FUNCTION LWORD_TO_QUARTERS
  (* Standard: 61499-1; Description: Copyright (c) 2024 HR Agrartechnik GmbH This program and the accompanying materials are made available under the terms of the Eclipse Public License 2.0 which is available at https://www.eclipse.org/legal/epl-2.0/ SPDX-License-Identifier: EPL-2.0 *)
  (* Version 1.0, 2024-02-22, franz *)
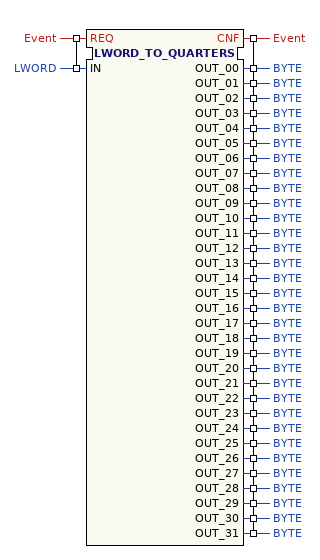
  EVENT_INPUT
    REQ WITH IN; (* Normal Execution Request *)
  END_EVENT
  EVENT_OUTPUT
    CNF WITH OUT_00, OUT_01, OUT_02, OUT_03, OUT_04, OUT_05, OUT_06, OUT_07, OUT_08, OUT_09, OUT_10, OUT_11, OUT_12, OUT_13, OUT_14, OUT_15, OUT_16, OUT_17, OUT_18, OUT_19, OUT_20, OUT_21, OUT_22, OUT_23, OUT_24, OUT_25, OUT_26, OUT_27, OUT_28, OUT_29, OUT_30, OUT_31; (* Execution Confirmation *)
  END_EVENT
  VAR_INPUT
    IN : LWORD; (* LWORD Input *)
  END_VAR
  VAR_OUTPUT
    OUT_00 : BYTE; (* QUARTER BYTE 00 *)
    OUT_01 : BYTE; (* QUARTER BYTE 01 *)
    OUT_02 : BYTE; (* QUARTER BYTE 02 *)
    OUT_03 : BYTE; (* QUARTER BYTE 03 *)
    OUT_04 : BYTE; (* QUARTER BYTE 04 *)
    OUT_05 : BYTE; (* QUARTER BYTE 05 *)
    OUT_06 : BYTE; (* QUARTER BYTE 06 *)
    OUT_07 : BYTE; (* QUARTER BYTE 07 *)
    OUT_08 : BYTE; (* QUARTER BYTE 08 *)
    OUT_09 : BYTE; (* QUARTER BYTE 09 *)
    OUT_10 : BYTE; (* QUARTER BYTE 10 *)
    OUT_11 : BYTE; (* QUARTER BYTE 11 *)
    OUT_12 : BYTE; (* QUARTER BYTE 12 *)
    OUT_13 : BYTE; (* QUARTER BYTE 13 *)
    OUT_14 : BYTE; (* QUARTER BYTE 14 *)
    OUT_15 : BYTE; (* QUARTER BYTE 15 *)
    OUT_16 : BYTE; (* QUARTER BYTE 16 *)
    OUT_17 : BYTE; (* QUARTER BYTE 17 *)
    OUT_18 : BYTE; (* QUARTER BYTE 18 *)
    OUT_19 : BYTE; (* QUARTER BYTE 19 *)
    OUT_20 : BYTE; (* QUARTER BYTE 20 *)
    OUT_21 : BYTE; (* QUARTER BYTE 21 *)
    OUT_22 : BYTE; (* QUARTER BYTE 22 *)
    OUT_23 : BYTE; (* QUARTER BYTE 23 *)
    OUT_24 : BYTE; (* QUARTER BYTE 24 *)
    OUT_25 : BYTE; (* QUARTER BYTE 25 *)
    OUT_26 : BYTE; (* QUARTER BYTE 26 *)
    OUT_27 : BYTE; (* QUARTER BYTE 27 *)
    OUT_28 : BYTE; (* QUARTER BYTE 28 *)
    OUT_29 : BYTE; (* QUARTER BYTE 29 *)
    OUT_30 : BYTE; (* QUARTER BYTE 30 *)
    OUT_31 : BYTE; (* QUARTER BYTE 31 *)
  END_VAR
  BODY IN ST:
FUNCTION LWORD_TO_QUARTERS

VAR_INPUT
	IN : LWORD;    // LWORD Input
END_VAR

VAR_OUTPUT
	OUT_00 : BYTE;    // QUARTER BYTE 00
	OUT_01 : BYTE;    // QUARTER BYTE 01
	OUT_02 : BYTE;    // QUARTER BYTE 02
	OUT_03 : BYTE;    // QUARTER BYTE 03
	OUT_04 : BYTE;    // QUARTER BYTE 04
	OUT_05 : BYTE;    // QUARTER BYTE 05
	OUT_06 : BYTE;    // QUARTER BYTE 06
	OUT_07 : BYTE;    // QUARTER BYTE 07
	OUT_08 : BYTE;    // QUARTER BYTE 08
	OUT_09 : BYTE;    // QUARTER BYTE 09
	OUT_10 : BYTE;    // QUARTER BYTE 10
	OUT_11 : BYTE;    // QUARTER BYTE 11
	OUT_12 : BYTE;    // QUARTER BYTE 12
	OUT_13 : BYTE;    // QUARTER BYTE 13
	OUT_14 : BYTE;    // QUARTER BYTE 14
	OUT_15 : BYTE;    // QUARTER BYTE 15
	OUT_16 : BYTE;    // QUARTER BYTE 16
	OUT_17 : BYTE;    // QUARTER BYTE 17
	OUT_18 : BYTE;    // QUARTER BYTE 18
	OUT_19 : BYTE;    // QUARTER BYTE 19
	OUT_20 : BYTE;    // QUARTER BYTE 20
	OUT_21 : BYTE;    // QUARTER BYTE 21
	OUT_22 : BYTE;    // QUARTER BYTE 22
	OUT_23 : BYTE;    // QUARTER BYTE 23
	OUT_24 : BYTE;    // QUARTER BYTE 24
	OUT_25 : BYTE;    // QUARTER BYTE 25
	OUT_26 : BYTE;    // QUARTER BYTE 26
	OUT_27 : BYTE;    // QUARTER BYTE 27
	OUT_28 : BYTE;    // QUARTER BYTE 28
	OUT_29 : BYTE;    // QUARTER BYTE 29
	OUT_30 : BYTE;    // QUARTER BYTE 30
	OUT_31 : BYTE;    // QUARTER BYTE 31
END_VAR

(* this Function extracts the 32 QUARTER BYTE from a lword *)
OUT_00 := LWORD_TO_BYTE(SHR(IN AND LWORD_QUARTER_00, SHFT_QUARTER_00));
OUT_01 := LWORD_TO_BYTE(SHR(IN AND LWORD_QUARTER_01, SHFT_QUARTER_01));
OUT_02 := LWORD_TO_BYTE(SHR(IN AND LWORD_QUARTER_02, SHFT_QUARTER_02));
OUT_03 := LWORD_TO_BYTE(SHR(IN AND LWORD_QUARTER_03, SHFT_QUARTER_03));
OUT_04 := LWORD_TO_BYTE(SHR(IN AND LWORD_QUARTER_04, SHFT_QUARTER_04));
OUT_05 := LWORD_TO_BYTE(SHR(IN AND LWORD_QUARTER_05, SHFT_QUARTER_05));
OUT_06 := LWORD_TO_BYTE(SHR(IN AND LWORD_QUARTER_06, SHFT_QUARTER_06));
OUT_07 := LWORD_TO_BYTE(SHR(IN AND LWORD_QUARTER_07, SHFT_QUARTER_07));
OUT_08 := LWORD_TO_BYTE(SHR(IN AND LWORD_QUARTER_08, SHIFT_QUARTER_08));
OUT_09 := LWORD_TO_BYTE(SHR(IN AND LWORD_QUARTER_09, SHIFT_QUARTER_09));
OUT_10 := LWORD_TO_BYTE(SHR(IN AND LWORD_QUARTER_10, SHIFT_QUARTER_10));
OUT_11 := LWORD_TO_BYTE(SHR(IN AND LWORD_QUARTER_11, SHIFT_QUARTER_11));
OUT_12 := LWORD_TO_BYTE(SHR(IN AND LWORD_QUARTER_12, SHIFT_QUARTER_12));
OUT_13 := LWORD_TO_BYTE(SHR(IN AND LWORD_QUARTER_13, SHIFT_QUARTER_13));
OUT_14 := LWORD_TO_BYTE(SHR(IN AND LWORD_QUARTER_14, SHIFT_QUARTER_14));
OUT_15 := LWORD_TO_BYTE(SHR(IN AND LWORD_QUARTER_15, SHIFT_QUARTER_15));
OUT_16 := LWORD_TO_BYTE(SHR(IN AND LWORD_QUARTER_16, SHIFT_QUARTER_16));
OUT_17 := LWORD_TO_BYTE(SHR(IN AND LWORD_QUARTER_17, SHIFT_QUARTER_17));
OUT_18 := LWORD_TO_BYTE(SHR(IN AND LWORD_QUARTER_18, SHIFT_QUARTER_18));
OUT_19 := LWORD_TO_BYTE(SHR(IN AND LWORD_QUARTER_19, SHIFT_QUARTER_19));
OUT_20 := LWORD_TO_BYTE(SHR(IN AND LWORD_QUARTER_20, SHIFT_QUARTER_20));
OUT_21 := LWORD_TO_BYTE(SHR(IN AND LWORD_QUARTER_21, SHIFT_QUARTER_21));
OUT_22 := LWORD_TO_BYTE(SHR(IN AND LWORD_QUARTER_22, SHIFT_QUARTER_22));
OUT_23 := LWORD_TO_BYTE(SHR(IN AND LWORD_QUARTER_23, SHIFT_QUARTER_23));
OUT_24 := LWORD_TO_BYTE(SHR(IN AND LWORD_QUARTER_24, SHIFT_QUARTER_24));
OUT_25 := LWORD_TO_BYTE(SHR(IN AND LWORD_QUARTER_25, SHIFT_QUARTER_25));
OUT_26 := LWORD_TO_BYTE(SHR(IN AND LWORD_QUARTER_26, SHIFT_QUARTER_26));
OUT_27 := LWORD_TO_BYTE(SHR(IN AND LWORD_QUARTER_27, SHIFT_QUARTER_27));
OUT_28 := LWORD_TO_BYTE(SHR(IN AND LWORD_QUARTER_28, SHIFT_QUARTER_28));
OUT_29 := LWORD_TO_BYTE(SHR(IN AND LWORD_QUARTER_29, SHIFT_QUARTER_29));
OUT_30 := LWORD_TO_BYTE(SHR(IN AND LWORD_QUARTER_30, SHIFT_QUARTER_30));
OUT_31 := LWORD_TO_BYTE(SHR(IN AND LWORD_QUARTER_31, SHIFT_QUARTER_31));

END_FUNCTION
  END_BODY
END_FUNCTION
